FUNCTION_BLOCK TEST_MUL (* Test MUL functions *)
  (* Standard: IEC 61499-1 *)
  (* Version 0.0, 2006-09-11, JHC, Holobloc Inc *)
  (* Compiler header: package fb.rt.test; *)
  (* Compiler classdef: SimpleFB *)
  (* Compiler Java Sun JDK 1.5.0 *)
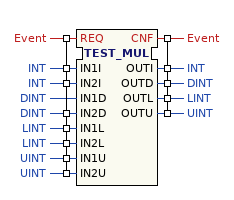
  EVENT_INPUT
    REQ WITH IN1I, IN2I, IN2D, IN1L, IN2L, IN1U, IN2U;
  END_EVENT
  EVENT_OUTPUT
    CNF WITH OUTI, OUTD, OUTL, OUTU;
  END_EVENT
  VAR_INPUT
    IN1I : INT;
    IN2I : INT;
    IN1D : DINT;
    IN2D : DINT;
    IN1L : LINT;
    IN2L : LINT;
    IN1U : UINT;
    IN2U : UINT;
  END_VAR
  VAR_OUTPUT
    OUTI : INT;
    OUTD : DINT;
    OUTL : LINT;
    OUTU : UINT;
  END_VAR
  ALGORITHM REQ IN FBD:
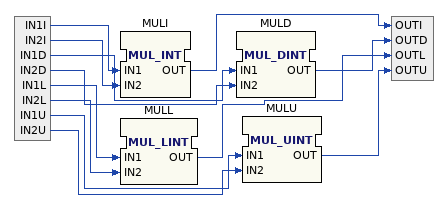
    FBS
      MULI : MUL_INT;
      MULD : MUL_DINT;
      MULL : MUL_LINT;
      MULU : MUL_UINT;
    END_FBS
    DATA_CONNECTIONS
      IN1I TO MULI.IN1;
      IN2I TO MULI.IN2;
      MULI.OUT TO OUTI;
      IN1D TO MULD.IN1;
      IN2D TO MULD.IN2;
      MULD.OUT TO OUTD;
      IN1L TO MULL.IN1;
      IN2L TO MULL.IN2;
      MULL.OUT TO OUTL;
      IN1U TO MULU.IN1;
      IN2U TO MULU.IN2;
      MULU.OUT TO OUTU;
    END_CONNECTIONS
  END_ALGORITHM
END_FUNCTION_BLOCK
